// TIA Portal V17 export
// export: Created 2023-12-22T15:28:38.1672159Z, ExportSetting WithDefaults, DisplayName Totally Integrated Automation Portal, DisplayVersion V17, DisplayName TIA Portal Openness, DisplayVersion V17, DisplayName TIA Portal Version Control Interface, DisplayVersion V17, DisplayName STEP 7 Professional, DisplayVersion V17, DisplayName STEP 7 Safety, DisplayVersion V17, DisplayName WinCC Advanced, DisplayVersion V17
TYPE "CMD"
// stored: IsFailsafeCompliant false
   STRUCT
      Start_A : Bool;   // Автозапуск / Запуск в авторежиме
      Start_M : Bool;   // Ручной - вперёд / Запуск в ручном режиме
      Hand : Bool;   // 0 - авто, 1 - ручной / 0 - Авто, 1 - Ручной
      Local : Bool;   // Локальный
      Lock : Bool;   // Блокировать / Блокировка
      Service : Bool;   // Сервис
      Safety : Bool;   // Безопасность
      Force : Bool;   // Принудительный
      Alarm : Bool;   // Есть авария / Авария
      Reset : Bool;   // Сброс аварий
      Sim : Bool;   // Режим симуляции
      Vector { S7_SetPoint := 'True'} : Bool;   // Выбор направления
      ResetOpTime : Bool;   // Сброс счётчика наработки
      Ready : Bool := true;   // Разрешение дистанционного управления
      reserv : Bool;
   END_STRUCT;
END_TYPE
